		IF DataFromPackML THEN
//			product					:= LREAL_TO_INT(_PackTags.Command.Parameter[2].Value);
//			PullWheels.Length		:= _PackTags.Command.Product[product].ProcessVariables[LENGTH].Value;
//			PullWheels.Velocity		:= _PackTags.Command.Product[product].ProcessVariables[PULLWHEELS_VEL].Value;
//			PullWheels.Acceleration := _PackTags.Command.Product[product].ProcessVariables[PULLWHEELS_ACC].Value;
//			Sealer.SealTime			:= _PackTags.Command.Product[product].ProcessVariables[SEALTIME].Value;
//			Sealer.Temp				:= _PackTags.Command.Product[product].ProcessVariables[SEALTEMP].Value;
//			Sealer.OpenPos			:= _PackTags.Command.Product[product].ProcessVariables[OPEN_POS].Value;
//			Sealer.ClosedPos		:= _PackTags.Command.Product[product].ProcessVariables[CLOSED_POS].Value;
//			Sealer.Velocity			:= _PackTags.Command.Product[product].ProcessVariables[SEALER_VEL].Value;
//			Sealer.Acceleration		:= _PackTags.Command.Product[product].ProcessVariables[SEALER_ACC].Value;
//			Unwind.Velocity			:= _PackTags.Command.Product[product].ProcessVariables[UNWIND_VEL].Value;
//			Unwind.Acceleration		:= _PackTags.Command.Product[product].ProcessVariables[UNWIND_ACC].Value;
		END_IF

	E_PMLUnitMode.ePMLUnitMode_Maintenance, E_PMLUnitMode.ePMLUnitMode_Manual:
		;
END_CASE

SUPER^.Resetting();
END_METHOD

METHOD PROTECTED Starting
VAR_INPUT
END_VAR
CASE _CurrentMode OF
	//=================================PRODUCTION MODE==================================
	E_PMLUnitMode.ePMLUnitMode_Production:
		// The seal bar can go to Execute, the others will be run in Mahcine Execute
	//	Sealer.Heat := TRUE;
		StateComplete();

	E_PMLUnitMode.ePMLUnitMode_Maintenance, E_PMLUnitMode.ePMLUnitMode_Manual:
		SUPER^.Starting();
END_CASE
END_METHOD

METHOD PROTECTED SubModuleMonitor : BOOL
VAR
	AlarmResponses : ARRAY[0..4] OF E_AlarmResponse; //Temporary response array	
END_VAR
// Check the sub Modules for Alarm Severity
SUPER^.SubModuleMonitor();

//Check the alarms at the machine level
_CurrentAlarmSeverity := F_GetMaxSeverityRaised(Alarms := MachineSafetyAlarms, CurrentSeverity := _CurrentAlarmSeverity);

//Check the severity of the machine level alarms
IF _CurrentState <> E_PMLState.ePMLState_Aborted AND _CurrentState <> E_PMLState.ePMLState_Aborting AND _CurrentState <> E_PMLState.ePMLState_Clearing AND _CurrentState <> E_PMLState.ePMLState_Stopped AND _CurrentState <> E_PMLState.ePMLState_Stopping THEN
	AlarmResponses := _ParentFaultResponseDefinitions;
	CASE AlarmResponses[CurrentAlarmSeverity] OF
		E_AlarmResponse.Abort_ImmediateError:
			AbortImmediateError(Name, TRUE);

		E_AlarmResponse.Abort_Immediate:
			AbortImmediate();

		E_AlarmResponse.Stop_Immediate:
			StopImmediate();

		E_AlarmResponse.Stop_Controlled:
			StopControlled();

		E_AlarmResponse.Hold_Immediate:
			HoldImmediate();

		E_AlarmResponse.Suspend_Immediate:
			SuspendImmediate();

		E_AlarmResponse.Suspend_Controlled:
			SuspendControlled();

		E_AlarmResponse.NoResponse:
			;
	END_CASE
ELSIF _CurrentState = E_PMLState.ePMLState_Stopped OR _CurrentState = E_PMLState.ePMLState_Stopping THEN
	AlarmResponses := _ParentFaultResponseDefinitions;
	CASE AlarmResponses[CurrentAlarmSeverity] OF
		E_AlarmResponse.Abort_ImmediateError:
			AbortImmediateError(Name, TRUE);

		E_AlarmResponse.Abort_Immediate:
			AbortImmediate();

		E_AlarmResponse.NoResponse:
			;
	END_CASE
END_IF
END_METHOD

METHOD PROTECTED Suspended
VAR_INPUT
END_VAR
//IF THIS^.Sealer.sealbar.InTempRange THEN
	ChangeState(E_PMLCommand.ePMLCommand_Unsuspend);
//END_IF
END_METHOD

METHOD PROTECTED Suspending
VAR_INPUT
END_VAR
CASE _CurrentMode OF
	//=================================PRODUCTION MODE==================================
	E_PMLUnitMode.ePMLUnitMode_Production:
	//	IF (Sealer.CurrentState = E_PMLState.ePMLState_Complete OR Sealer.CurrentState = E_PMLState.ePMLState_Idle) AND (PullWheels.CurrentState = E_PMLState.ePMLState_Complete OR PullWheels.CurrentState = E_PMLState.ePMLState_Idle) THEN
			StateComplete();
	//	END_IF

	E_PMLUnitMode.ePMLUnitMode_Maintenance, E_PMLUnitMode.ePMLUnitMode_Manual:
		SUPER^.Suspending();
END_CASE
END_METHOD

METHOD PROTECTED Unholding
VAR_INPUT
END_VAR
CASE _CurrentMode OF
	//=================================PRODUCTION MODE==================================
	E_PMLUnitMode.ePMLUnitMode_Production:
		StateComplete();

	E_PMLUnitMode.ePMLUnitMode_Maintenance, E_PMLUnitMode.ePMLUnitMode_Manual:
		SUPER^.Unholding();
END_CASE
END_METHOD

METHOD PROTECTED Unsuspending
VAR_INPUT
END_VAR
CASE _CurrentMode OF
	//=================================PRODUCTION MODE==================================
	E_PMLUnitMode.ePMLUnitMode_Production:
		StateComplete();

	E_PMLUnitMode.ePMLUnitMode_Maintenance, E_PMLUnitMode.ePMLUnitMode_Manual:
		SUPER^.Unsuspending();
END_CASE
END_METHOD

METHOD UpdateModeTimers
VAR
	currentTime	 : T_DCTIME64;
	timeToUpdate : LREAL;
END_VAR

VAR_INST
	lastTime  : T_DCTIME64 := F_GetActualDcTime64();
	lastState : DINT;
	lastMode  : DINT;
END_VAR
IF _PackTags.Status.StateCurrent <> lastState THEN
	MEMSET(ADR(_PackTags.Admin.StateCurrentTime), 0, SIZEOF(_PackTags.Admin.StateCurrentTime));
	lastState := _PackTags.Status.StateCurrent;
END_IF

IF _PackTags.Status.UnitModeCurrent <> lastMode THEN
	MEMSET(ADR(_PackTags.Admin.ModeCurrentTime), 0, SIZEOF(_PackTags.Admin.ModeCurrentTime));
	lastMode := _PackTags.Status.UnitModeCurrent;
END_IF

currentTime := F_GetActualDcTime64();
IF lastTime <> 0 THEN
	timeToUpdate := ULINT_TO_LREAL(currentTime - lastTime) / 1_000_000_000.0;
END_IF

// only seconds get added to the cumulative timers 
IF timeToUpdate > 1 THEN
	_PackTags.Admin.ModeCummulativeTime[_PackTags.Status.UnitModeCurrent]								  := _PackTags.Admin.ModeCummulativeTime[_PackTags.Status.UnitModeCurrent] + LREAL_TO_DINT(timeToUpdate);
	_PackTags.Admin.ModeCurrentTime[_PackTags.Status.UnitModeCurrent]									  := _PackTags.Admin.ModeCurrentTime[_PackTags.Status.UnitModeCurrent] + LREAL_TO_DINT(timeToUpdate);
	_PackTags.Admin.StateCummulativeTime[_PackTags.Status.UnitModeCurrent, _PackTags.Status.StateCurrent] := _PackTags.Admin.StateCummulativeTime[_PackTags.Status.UnitModeCurrent, _PackTags.Status.StateCurrent] + LREAL_TO_DINT(timeToUpdate);
	_PackTags.Admin.StateCurrentTime[_PackTags.Status.UnitModeCurrent, _PackTags.Status.StateCurrent]	  := _PackTags.Admin.StateCurrentTime[_PackTags.Status.UnitModeCurrent, _PackTags.Status.StateCurrent] + LREAL_TO_DINT(timeToUpdate);
	lastTime																							  := currentTime;
END_IF
END_METHOD

END_FUNCTION_BLOCK

// ---- Machine/FB_Systems.TcPOU
FUNCTION_BLOCK FB_Systems EXTENDS FB_PackML_BaseModule // IMPLEMENTS I_ControlsProductionRate
VAR
	// Sub Modules

	
//	Safety			: FB_Safety_Module			:= (Name := 'Safety', LogStateChanges := TRUE);
	Diagnostics		: FB_Diagnostics_Module		:= (Name := 'Diagnostics', LogStateChanges := TRUE);


	// Components

	//Initial List of Components
	ipComponents_Init : ARRAY[1..Parameters_PackML_Base.MAX_NO_OF_COMPONENTS] OF I_ComponentBase := [];

	//Alarms for this module
	SystemAlarms : ARRAY[1..SYTEM_ALARM_COUNT] OF FB_TcAlarm;

	//Current Recipe Name
	CurrentRecipeName : STRING;

	//Get Data From PackML? Else RecipeManager is running
	DataFromPackML : BOOL := TRUE;

	//Data 
	sealTimeStart : ULINT;
	sealTimeEnd	  : ULINT;
	sealingTime	  : LREAL;
	sealTrig	  : R_TRIG;
	pullTimeStart : ULINT;
	pullTimeEnd	  : ULINT;
	pullingTime	  : LREAL;
	pulltrig	  : R_TRIG;
	partTimeStart : ULINT;
	partTimeEnd	  : ULINT;
	partTime	  : LREAL;
	parts		  : DINT;
	product		  : DINT;

	//Pack Tags for System
	{attribute 'OPC.UA.DA' := '1'}
	_PackTags : ST_PackMLv30Ext; //ST_PackMLv30 is obsolete in Tc3_PackML_V2
END_VAR

VAR CONSTANT
	//PackTag parameter IDs
	LENGTH		   : INT := 1;
	SEALTEMP	   : INT := 2;
	SEALTIME	   : INT := 3;
	PULLWHEELS_VEL : INT := 4;
	PULLWHEELS_ACC : INT := 5;
	SEALER_VEL	   : INT := 6;
	SEALER_ACC	   : INT := 7;
	UNWIND_VEL	   : INT := 8;
	UNWIND_ACC	   : INT := 9;
	OPEN_POS	   : INT := 10;
	CLOSED_POS	   : INT := 11;

	//Alarm count constant
	SYTEM_ALARM_COUNT : INT := 6;
END_VAR

// Simulation variables
VAR
	EstopInput	: BOOL;
	LowAirInput : BOOL;
	ErrorInput	: BOOL;
	WarnInput	: BOOL;
	InfoInput	: BOOL;
END_VAR

//This needs to go straight to run mode I did this on the turbine modules
//Stuff for this module
//Maintenance monitoring.
//System communication - Azure - API
//							MQTT
//System times

METHOD PROTECTED Completing
VAR_INPUT
END_VAR
CASE _CurrentMode OF
	//=================================PRODUCTION MODE==================================
	E_PMLUnitMode.ePMLUnitMode_Production:
		StateComplete();

	E_PMLUnitMode.ePMLUnitMode_Maintenance, E_PMLUnitMode.ePMLUnitMode_Manual:
		SUPER^.Completing();
END_CASE
END_METHOD

METHOD PROTECTED CreateEvents
VAR_INPUT
END_VAR
// Add your event creation here
F_CreateAllEventsInClass(Alarms		:= SystemAlarms,
						 ClassSize	:= SIZEOF(TC_Events.VFFSDemo),
						 pInitEvent := ADR(TC_EVENTS.VFFSDemo.InitReferenceEvent),
						 Prefix		:= Name);

// Super call to base
SUPER^.CreateEvents();
END_METHOD

METHOD CyclicLogic
VAR_INPUT
END_VAR
IF NOT _InitComplete THEN
	_InitComplete := Initialize();
	RETURN;
END_IF

SUPER^.CyclicLogic();

// Fill in the PackTags for the machine output
_PackTags.Status.StateCurrent	 := _CurrentState;
_PackTags.Status.UnitModeCurrent := _CurrentMode;
UpdateModeTimers();

//This is just to simulate some IO for alarms
//CyclicLogic_Simulation();
END_METHOD

METHOD CyclicLogic_Simulation
VAR_INPUT
END_VAR

VAR_INST
END_VAR
(*	
This is just for testing. Real hardware can be setup in other places
Here the alarms will raise and clear on its own if the input changes	
*)
IF EstopInput AND NOT MachineAlarms[E_VFFSDemo.EmergencyStop].bRaised THEN
	RaiseAlarm2Args(MachineAlarms[E_VFFSDemo.EmergencyStop], '', '');
ELSIF NOT EstopInput AND MachineAlarms[E_VFFSDemo.EmergencyStop].bRaised THEN
	MachineAlarms[E_VFFSDemo.EmergencyStop].Clear(0, 0);
END_IF

IF LowAirInput AND NOT MachineAlarms[E_VFFSDemo.LowAir].bRaised THEN
	RaiseAlarm2Args(MachineAlarms[E_VFFSDemo.LowAir], '', '');
ELSIF NOT LowAirInput AND MachineAlarms[E_VFFSDemo.LowAir].bRaised THEN
	MachineAlarms[E_VFFSDemo.LowAir].Clear(0, 0);
END_IF

//Generic Alarms for Testing
IF ErrorInput AND NOT MachineAlarms[E_VFFSDemo.AlarmMessage].bRaised THEN
	RaiseAlarm2Args(MachineAlarms[E_VFFSDemo.AlarmMessage], '', '');
ELSIF NOT ErrorInput AND MachineAlarms[E_VFFSDemo.AlarmMessage].bRaised THEN
	MachineAlarms[E_VFFSDemo.AlarmMessage].Clear(0, 0);
END_IF

IF WarnInput AND NOT MachineAlarms[E_VFFSDemo.WarnMessage].bRaised THEN
	RaiseAlarm2Args(MachineAlarms[E_VFFSDemo.WarnMessage], '', '');
ELSIF NOT WarnInput AND MachineAlarms[E_VFFSDemo.WarnMessage].bRaised THEN
	MachineAlarms[E_VFFSDemo.WarnMessage].Clear(0, 0);
END_IF

IF InfoInput AND NOT MachineAlarms[E_VFFSDemo.InfoMessage].bRaised THEN
	RaiseAlarm2Args(MachineAlarms[E_VFFSDemo.InfoMessage], '', '');
ELSIF NOT InfoInput AND MachineAlarms[E_VFFSDemo.InfoMessage].bRaised THEN
	MachineAlarms[E_VFFSDemo.InfoMessage].Clear(0, 0);
END_IF
END_METHOD

METHOD PROTECTED FINAL Execute
VAR_INPUT
END_VAR
CASE _CurrentMode OF
	//=================================PRODUCTION MODE==================================
	E_PMLUnitMode.ePMLUnitMode_Production:
		(* Run the sequence to make products 
		 Unwind Runs Slowly 
		 Pull Wheels Run 
		 Jaws Seal, and Repeat until production reached*)
		sealTrig(CLK := SequenceState = 10);
		IF sealTrig.Q THEN
			partTimeStart := F_GetActualDcTime64();
			sealTimeStart := partTimeStart;
		END_IF

		pulltrig(CLK := SequenceState = 20);
		IF pulltrig.Q THEN
			pullTimeStart := F_GetActualDcTime64();
		END_IF

//		IF THIS^.Sealer.sealbar.InTempRange THEN
//			CASE SequenceState OF
//				0: //Started
//					Unwind.ChangeState(E_PMLCommand.ePMLCommand_Start);
//					IF Unwind.CurrentState = E_PMLState.ePMLState_Execute THEN
//						SequenceState := SequenceState + 10;
//					END_IF

//				10: // SEAL First
//					Sealer.ChangeState(E_PMLCommand.ePMLCommand_Start);
//					IF Sealer.CurrentState = E_PMLState.ePMLState_Complete THEN
//						Sealer.ChangeState(E_PMLCommand.ePMLCommand_Reset);
//						SequenceState := SequenceState + 10;
//						SealTimeEnd	  := F_GetActualDcTime64();
//						sealingTime	  := ULINT_TO_LREAL(sealtimeEnd - sealTimeStart) * 1E-9;
//					END_IF

//				20: // Run Pullwheels
//					PullWheels.ChangeState(E_PMLCommand.ePMLCommand_Start);
//					IF PullWheels.CurrentState = E_PMLState.ePMLState_Complete THEN
//						partTimeEnd	  := F_GetActualDcTime64();
//						parts		  := parts + 1;
//						SequenceState := 10;
//						PullWheels.ChangeState(E_PMLCommand.ePMLCommand_Reset);
//						pullTimeEnd := F_GetActualDcTime64();
//						pullingTime := ULINT_TO_LREAL(pullTimeEnd - pullTimeStart) * 1E-9;
//					END_IF
//			END_CASE
//		ELSE
//			ChangeState(E_PMLCommand.ePMLCommand_Suspend);
//		END_IF

	//=================================MAINTENANCE MODE==================================	
	E_PMLUnitMode.ePMLUnitMode_Maintenance:
		;

	//=================================MANUAL MODE==================================
	E_PMLUnitMode.ePMLUnitMode_Manual:
		;
END_CASE
END_METHOD

METHOD PROTECTED Held
VAR_INPUT
END_VAR
END_METHOD

METHOD PROTECTED HMIPermissions
VAR_INPUT
END_VAR
//General Mode Based Monitoring and handling of HMI control
CASE _CurrentMode OF
	E_PMLUnitMode.ePMLUnitMode_Production:
		CASE _CurrentState OF
			E_PMLState.ePMLState_Stopped:
				AllowHMIControl(ThisModuleOnly := TRUE); //Allow control for recovery
			E_PMLState.ePMLState_Idle:
				//BlockHMIControl();
				AllowHMIControl(ThisModuleOnly := TRUE); //Allow control for recovery
			E_PMLState.ePMLState_Suspended:
				BlockHMIControl();

			E_PMLState.ePMLState_Execute:
				BlockHMIControl();

			E_PMLState.ePMLState_Aborted:
				AllowHMIControl(ThisModuleOnly := TRUE); //Allow control for recovery
			E_PMLState.ePMLState_Held:
				AllowHMIControl(ThisModuleOnly := TRUE); //Allow control for recovery
			E_PMLState.ePMLState_Complete:
				BlockHMIControl();
		END_CASE

	//AllowHMIControl(ThisModuleOnly := FALSE);
	E_PMLUnitMode.ePMLUnitMode_Manual:
		AllowHMIControl(ThisModuleOnly := FALSE);

	E_PMLUnitMode.ePMLUnitMode_Maintenance:
		AllowHMIControl(ThisModuleOnly := FALSE);
END_CASE
END_METHOD

METHOD PROTECTED HoldImmediate
VAR_INPUT
END_VAR
ChangeState(E_PMLCommand.ePMLCommand_Hold);
END_METHOD

METHOD PROTECTED Holding
VAR_INPUT
END_VAR
CASE _CurrentMode OF
	//=================================PRODUCTION MODE==================================
	E_PMLUnitMode.ePMLUnitMode_Production:
	//	IF (Sealer.CurrentState = E_PMLState.ePMLState_Complete OR Sealer.CurrentState = E_PMLState.ePMLState_Idle) AND (PullWheels.CurrentState = E_PMLState.ePMLState_Complete OR PullWheels.CurrentState = E_PMLState.ePMLState_Idle) THEN
			StateComplete();
	//	END_IF

	E_PMLUnitMode.ePMLUnitMode_Maintenance, E_PMLUnitMode.ePMLUnitMode_Manual:
		SUPER^.Holding();
END_CASE
END_METHOD

METHOD PROTECTED Initialize : BOOL
VAR
	i : UDINT; //Generic iteration value
END_VAR
Initialize := FALSE;
CASE DescendantSequenceState OF
	0:
//		RegisterSubmodule(PullWheels);
//		RegisterSubmodule(Sealer);
//		RegisterSubmodule(Unwind);
		
//		RegisterSubmodule(Safety);
		RegisterSubmodule(Diagnostics);
//		RegisterSubmodule(Closer_Gluer);
//		RegisterSubmodule(Labeler);
//		RegisterSubmodule(Diverter);
//		RegisterSubmodule(Outfeed);
		
		_LogModeChanges			:= FALSE;
		_LogStateChanges		:= FALSE;
		DescendantSequenceState := DescendantSequenceState + 10;

	10:
		//Setup Custom modes here

		(*CustomModes(eMode                          :=,
                    sName                          :=,
                    bDisableClearing               :=,
                    bDisableStarting               :=,
                    bDisableSuspended              :=,
                    bDisableStopping               :=,
                    bDisableAborting               :=,
                    bDisableHolding                :=,
                    bDisableHeld                   :=,
                    bDisableUnholding              :=,
                    bDisableSuspending             :=,
                    bDisableUnsuspending           :=,
                    bDisableResetting              :=,
                    bDisableIdle                   :=,
                    bDisableCompleting             :=,
                    bDisableComplete               :=,
                    bEnableUnitModeChangeStopped   :=,
                    bEnableUnitModeChangeIdle      :=,
                    bEnableUnitModeChangeSuspended :=,
                    bEnableUnitModeChangeExecute   :=,
                    bEnableUnitModeChangeAborted   :=,
                    bEnableUnitModeChangeHeld      :=,
                    bEnableUnitModeChangeComplete  :=,
                    bError                         =>,
                    nErrorId                       =>);*)
		DescendantSequenceState := DescendantSequenceState + 10;

	20:
		//Copy Mode names
		FOR i := 1 TO 3 DO
			ModeNames[i] := F_UnitModeToString(UDINT_TO_DINT(i));
		END_FOR

		DescendantSequenceState := DescendantSequenceState + 10;

	30:
		// Initialize Recipes 
		Initialize_Recipes();
		DescendantSequenceState := DescendantSequenceState + 10;

	40:
		//Call the Super
		IF SUPER^.Initialize() THEN
			DescendantSequenceState := DescendantSequenceState + 10;
		END_IF

	50:
		Initialize := TRUE;
END_CASE
END_METHOD

METHOD Initialize_Recipes
VAR_INPUT
END_VAR
// configuration of parameters Max Speed
_packTags.Command.Parameter[1].ID	 := 1;
_packTags.Command.Parameter[1].Name	 := 'Max Speed';
_packTags.Command.Parameter[1].Unit	 := '/min';
_packTags.Command.Parameter[1].Value := 180;
_packTags.Command.Parameter[2].ID	 := 2;
_packTags.Command.Parameter[2].Name	 := 'Product to Run';
_packTags.Command.Parameter[2].Unit	 := '';
_packTags.Command.Parameter[2].Value := 1;

// Recipe Product 1
_PackTags.Command.Product[1].ProductID								:= 100;
_PackTags.Command.Product[1].Ingredients[1].IngredientID			:= 1;
_PackTags.Command.Product[1].Ingredients[1].Parameter[1].ID			:= _PackTags.Command.Product[1].ProductID * 10 + 1;
_PackTags.Command.Product[1].Ingredients[1].Parameter[1].Name		:= 'Material Type';
_PackTags.Command.Product[1].Ingredients[1].Parameter[1].Unit		:= 'n/a';
_PackTags.Command.Product[1].Ingredients[1].Parameter[1].Value		:= 5;
_PackTags.Command.Product[1].Ingredients[1].Parameter[2].ID			:= _PackTags.Command.Product[1].ProductID * 10 + 2;
_PackTags.Command.Product[1].Ingredients[1].Parameter[2].Name		:= 'Material Thickness';
_PackTags.Command.Product[1].Ingredients[1].Parameter[2].Unit		:= 'um';
_PackTags.Command.Product[1].Ingredients[1].Parameter[2].Value		:= 240;
_PackTags.Command.Product[1].ProcessVariables[LENGTH].ID			:= _PackTags.Command.Product[1].ProductID * 20 + 1;
_PackTags.Command.Product[1].ProcessVariables[LENGTH].Name			:= 'Length';
_PackTags.Command.Product[1].ProcessVariables[LENGTH].Unit			:= 'mm';
_PackTags.Command.Product[1].ProcessVariables[LENGTH].Value			:= 100;
_PackTags.Command.Product[1].ProcessVariables[SEALTEMP].ID			:= _PackTags.Command.Product[1].ProductID * 20 + 2;
_PackTags.Command.Product[1].ProcessVariables[SEALTEMP].Name		:= 'Sealing Temp';
_PackTags.Command.Product[1].ProcessVariables[SEALTEMP].Unit		:= 'C';
_PackTags.Command.Product[1].ProcessVariables[SEALTEMP].Value		:= 100;
_PackTags.Command.Product[1].ProcessVariables[SEALTIME].ID			:= _PackTags.Command.Product[1].ProductID * 20 + 3;
_PackTags.Command.Product[1].ProcessVariables[SEALTIME].Name		:= 'Sealing Time';
_PackTags.Command.Product[1].ProcessVariables[SEALTIME].Unit		:= 'ms';
_PackTags.Command.Product[1].ProcessVariables[SEALTIME].Value		:= 50;
_PackTags.Command.Product[1].ProcessVariables[PULLWHEELS_VEL].ID	:= _PackTags.Command.Product[1].ProductID * 20 + 4;
_PackTags.Command.Product[1].ProcessVariables[PULLWHEELS_VEL].Name	:= 'Pull Wheels Vel';
_PackTags.Command.Product[1].ProcessVariables[PULLWHEELS_VEL].Unit	:= 'mm/s';
_PackTags.Command.Product[1].ProcessVariables[PULLWHEELS_VEL].Value := 100;
_PackTags.Command.Product[1].ProcessVariables[PULLWHEELS_ACC].ID	:= _PackTags.Command.Product[1].ProductID * 20 + 5;
_PackTags.Command.Product[1].ProcessVariables[PULLWHEELS_ACC].Name	:= 'Pull Wheels Acc';
_PackTags.Command.Product[1].ProcessVariables[PULLWHEELS_ACC].Unit	:= 'mm/s2';
_PackTags.Command.Product[1].ProcessVariables[PULLWHEELS_ACC].Value := 1000;
_PackTags.Command.Product[1].ProcessVariables[OPEN_POS].ID			:= _PackTags.Command.Product[1].ProductID * 20 + 6;
_PackTags.Command.Product[1].ProcessVariables[OPEN_POS].Name		:= 'Sealer Open Position';
_PackTags.Command.Product[1].ProcessVariables[OPEN_POS].Unit		:= 'mm';
_PackTags.Command.Product[1].ProcessVariables[OPEN_POS].Value		:= 105;
_PackTags.Command.Product[1].ProcessVariables[CLOSED_POS].ID		:= _PackTags.Command.Product[1].ProductID * 20 + 7;
_PackTags.Command.Product[1].ProcessVariables[CLOSED_POS].Name		:= 'Sealer Closed Position';
_PackTags.Command.Product[1].ProcessVariables[CLOSED_POS].Unit		:= 'mm';
_PackTags.Command.Product[1].ProcessVariables[CLOSED_POS].Value		:= 250;
_PackTags.Command.Product[1].ProcessVariables[SEALER_VEL].ID		:= _PackTags.Command.Product[1].ProductID * 20 + 8;
_PackTags.Command.Product[1].ProcessVariables[SEALER_VEL].Name		:= 'Sealer Vel';
_PackTags.Command.Product[1].ProcessVariables[SEALER_VEL].Unit		:= 'mm/s';
_PackTags.Command.Product[1].ProcessVariables[SEALER_VEL].Value		:= 100;
_PackTags.Command.Product[1].ProcessVariables[SEALER_ACC].ID		:= _PackTags.Command.Product[1].ProductID * 20 + 9;
_PackTags.Command.Product[1].ProcessVariables[SEALER_ACC].Name		:= 'Sealer Acc';
_PackTags.Command.Product[1].ProcessVariables[SEALER_ACC].Unit		:= 'mm/s2';
_PackTags.Command.Product[1].ProcessVariables[SEALER_ACC].Value		:= 1000;
_PackTags.Command.Product[1].ProcessVariables[UNWIND_VEL].ID		:= _PackTags.Command.Product[1].ProductID * 20 + 10;
_PackTags.Command.Product[1].ProcessVariables[UNWIND_VEL].Name		:= 'Unwind Vel';
_PackTags.Command.Product[1].ProcessVariables[UNWIND_VEL].Unit		:= 'mm/s';
_PackTags.Command.Product[1].ProcessVariables[UNWIND_VEL].Value		:= 100;
_PackTags.Command.Product[1].ProcessVariables[UNWIND_ACC].ID		:= _PackTags.Command.Product[1].ProductID * 20 + 11;
_PackTags.Command.Product[1].ProcessVariables[UNWIND_ACC].Name		:= 'Unwind Acc';
_PackTags.Command.Product[1].ProcessVariables[UNWIND_ACC].Unit		:= 'mm/s2';
_PackTags.Command.Product[1].ProcessVariables[UNWIND_ACC].Value		:= 1000;

// Product 2
_PackTags.Command.Product[2].ProductID								:= 100;
_PackTags.Command.Product[2].Ingredients[1].IngredientID			:= 1;
_PackTags.Command.Product[2].Ingredients[1].Parameter[1].ID			:= _PackTags.Command.Product[1].ProductID * 10 + 1;
_PackTags.Command.Product[2].Ingredients[1].Parameter[1].Name		:= 'Material Type';
_PackTags.Command.Product[2].Ingredients[1].Parameter[1].Unit		:= 'n/a';
_PackTags.Command.Product[2].Ingredients[1].Parameter[1].Value		:= 2;
_PackTags.Command.Product[2].Ingredients[1].Parameter[2].ID			:= _PackTags.Command.Product[1].ProductID * 10 + 2;
_PackTags.Command.Product[2].Ingredients[1].Parameter[2].Name		:= 'Material Thickness';
_PackTags.Command.Product[2].Ingredients[1].Parameter[2].Unit		:= 'um';
_PackTags.Command.Product[2].Ingredients[1].Parameter[2].Value		:= 220;
_PackTags.Command.Product[2].ProcessVariables[LENGTH].ID			:= _PackTags.Command.Product[1].ProductID * 20 + 1;
_PackTags.Command.Product[2].ProcessVariables[LENGTH].Name			:= 'Length';
_PackTags.Command.Product[2].ProcessVariables[LENGTH].Unit			:= 'mm';
_PackTags.Command.Product[2].ProcessVariables[LENGTH].Value			:= 55;
_PackTags.Command.Product[2].ProcessVariables[SEALTEMP].ID			:= _PackTags.Command.Product[1].ProductID * 20 + 2;
_PackTags.Command.Product[2].ProcessVariables[SEALTEMP].Name		:= 'Sealing Temp';
_PackTags.Command.Product[2].ProcessVariables[SEALTEMP].Unit		:= 'C';
_PackTags.Command.Product[2].ProcessVariables[SEALTEMP].Value		:= 110;
_PackTags.Command.Product[2].ProcessVariables[SEALTIME].ID			:= _PackTags.Command.Product[1].ProductID * 20 + 3;
_PackTags.Command.Product[2].ProcessVariables[SEALTIME].Name		:= 'Sealing Time';
_PackTags.Command.Product[2].ProcessVariables[SEALTIME].Unit		:= 'ms';
_PackTags.Command.Product[2].ProcessVariables[SEALTIME].Value		:= 100;
_PackTags.Command.Product[2].ProcessVariables[PULLWHEELS_VEL].ID	:= _PackTags.Command.Product[1].ProductID * 20 + 4;
_PackTags.Command.Product[2].ProcessVariables[PULLWHEELS_VEL].Name	:= 'Pull Wheels Vel';
_PackTags.Command.Product[2].ProcessVariables[PULLWHEELS_VEL].Unit	:= 'mm/s';
_PackTags.Command.Product[2].ProcessVariables[PULLWHEELS_VEL].Value := 200;
_PackTags.Command.Product[2].ProcessVariables[PULLWHEELS_ACC].ID	:= _PackTags.Command.Product[1].ProductID * 20 + 5;
_PackTags.Command.Product[2].ProcessVariables[PULLWHEELS_ACC].Name	:= 'Pull Wheels Acc';
_PackTags.Command.Product[2].ProcessVariables[PULLWHEELS_ACC].Unit	:= 'mm/s2';
_PackTags.Command.Product[2].ProcessVariables[PULLWHEELS_ACC].Value := 2000;
_PackTags.Command.Product[2].ProcessVariables[OPEN_POS].ID			:= _PackTags.Command.Product[1].ProductID * 20 + 6;
_PackTags.Command.Product[2].ProcessVariables[OPEN_POS].Name		:= 'Sealer Open Position';
_PackTags.Command.Product[2].ProcessVariables[OPEN_POS].Unit		:= 'mm';
_PackTags.Command.Product[2].ProcessVariables[OPEN_POS].Value		:= 60;
_PackTags.Command.Product[2].ProcessVariables[CLOSED_POS].ID		:= _PackTags.Command.Product[1].ProductID * 20 + 7;
_PackTags.Command.Product[2].ProcessVariables[CLOSED_POS].Name		:= 'Sealer Closed Position';
_PackTags.Command.Product[2].ProcessVariables[CLOSED_POS].Unit		:= 'mm';
_PackTags.Command.Product[2].ProcessVariables[CLOSED_POS].Value		:= 253;
_PackTags.Command.Product[2].ProcessVariables[SEALER_VEL].ID		:= _PackTags.Command.Product[1].ProductID * 20 + 8;
_PackTags.Command.Product[2].ProcessVariables[SEALER_VEL].Name		:= 'Sealer Vel';
_PackTags.Command.Product[2].ProcessVariables[SEALER_VEL].Unit		:= 'mm/s';
_PackTags.Command.Product[2].ProcessVariables[SEALER_VEL].Value		:= 200;
_PackTags.Command.Product[2].ProcessVariables[SEALER_ACC].ID		:= _PackTags.Command.Product[1].ProductID * 20 + 9;
_PackTags.Command.Product[2].ProcessVariables[SEALER_ACC].Name		:= 'Sealer Acc';
_PackTags.Command.Product[2].ProcessVariables[SEALER_ACC].Unit		:= 'mm/s2';
_PackTags.Command.Product[2].ProcessVariables[SEALER_ACC].Value		:= 2000;
_PackTags.Command.Product[2].ProcessVariables[UNWIND_VEL].ID		:= _PackTags.Command.Product[1].ProductID * 20 + 10;
_PackTags.Command.Product[2].ProcessVariables[UNWIND_VEL].Name		:= 'Unwind Vel';
_PackTags.Command.Product[2].ProcessVariables[UNWIND_VEL].Unit		:= 'mm/s';
_PackTags.Command.Product[2].ProcessVariables[UNWIND_VEL].Value		:= 200;
_PackTags.Command.Product[2].ProcessVariables[UNWIND_ACC].ID		:= _PackTags.Command.Product[1].ProductID * 20 + 11;
_PackTags.Command.Product[2].ProcessVariables[UNWIND_ACC].Name		:= 'Unwind Acc';
_PackTags.Command.Product[2].ProcessVariables[UNWIND_ACC].Unit		:= 'mm/s2';
_PackTags.Command.Product[2].ProcessVariables[UNWIND_ACC].Value		:= 2000;

//Product 3
_PackTags.Command.Product[3].ProductID								:= 307;
_PackTags.Command.Product[3].Ingredients[1].IngredientID			:= 1;
_PackTags.Command.Product[3].Ingredients[1].Parameter[1].ID			:= _PackTags.Command.Product[1].ProductID * 10 + 1;
_PackTags.Command.Product[3].Ingredients[1].Parameter[1].Name		:= 'Material Type';
_PackTags.Command.Product[3].Ingredients[1].Parameter[1].Unit		:= 'n/a';
_PackTags.Command.Product[3].Ingredients[1].Parameter[1].Value		:= 2;
_PackTags.Command.Product[3].Ingredients[1].Parameter[2].ID			:= _PackTags.Command.Product[1].ProductID * 10 + 2;
_PackTags.Command.Product[3].Ingredients[1].Parameter[2].Name		:= 'Material Thickness';
_PackTags.Command.Product[3].Ingredients[1].Parameter[2].Unit		:= 'um';
_PackTags.Command.Product[3].Ingredients[1].Parameter[2].Value		:= 220;
_PackTags.Command.Product[3].ProcessVariables[LENGTH].ID			:= _PackTags.Command.Product[1].ProductID * 20 + 1;
_PackTags.Command.Product[3].ProcessVariables[LENGTH].Name			:= 'Length';
_PackTags.Command.Product[3].ProcessVariables[LENGTH].Unit			:= 'mm';
_PackTags.Command.Product[3].ProcessVariables[LENGTH].Value			:= 85;
_PackTags.Command.Product[3].ProcessVariables[SEALTEMP].ID			:= _PackTags.Command.Product[1].ProductID * 20 + 2;
_PackTags.Command.Product[3].ProcessVariables[SEALTEMP].Name		:= 'Sealing Temp';
_PackTags.Command.Product[3].ProcessVariables[SEALTEMP].Unit		:= 'C';
_PackTags.Command.Product[3].ProcessVariables[SEALTEMP].Value		:= 95;
_PackTags.Command.Product[3].ProcessVariables[SEALTIME].ID			:= _PackTags.Command.Product[1].ProductID * 20 + 3;
_PackTags.Command.Product[3].ProcessVariables[SEALTIME].Name		:= 'Sealing Time';
_PackTags.Command.Product[3].ProcessVariables[SEALTIME].Unit		:= 'ms';
_PackTags.Command.Product[3].ProcessVariables[SEALTIME].Value		:= 20;
_PackTags.Command.Product[3].ProcessVariables[PULLWHEELS_VEL].ID	:= _PackTags.Command.Product[1].ProductID * 20 + 4;
_PackTags.Command.Product[3].ProcessVariables[PULLWHEELS_VEL].Name	:= 'Pull Wheels Vel';
_PackTags.Command.Product[3].ProcessVariables[PULLWHEELS_VEL].Unit	:= 'mm/s';
_PackTags.Command.Product[3].ProcessVariables[PULLWHEELS_VEL].Value := 300;
_PackTags.Command.Product[3].ProcessVariables[PULLWHEELS_ACC].ID	:= _PackTags.Command.Product[1].ProductID * 20 + 5;
_PackTags.Command.Product[3].ProcessVariables[PULLWHEELS_ACC].Name	:= 'Pull Wheels Acc';
_PackTags.Command.Product[3].ProcessVariables[PULLWHEELS_ACC].Unit	:= 'mm/s2';
_PackTags.Command.Product[3].ProcessVariables[PULLWHEELS_ACC].Value := 3000;
_PackTags.Command.Product[3].ProcessVariables[OPEN_POS].ID			:= _PackTags.Command.Product[1].ProductID * 20 + 6;
_PackTags.Command.Product[3].ProcessVariables[OPEN_POS].Name		:= 'Sealer Open Position';
_PackTags.Command.Product[3].ProcessVariables[OPEN_POS].Unit		:= 'mm';
_PackTags.Command.Product[3].ProcessVariables[OPEN_POS].Value		:= 56;
_PackTags.Command.Product[3].ProcessVariables[CLOSED_POS].ID		:= _PackTags.Command.Product[1].ProductID * 20 + 7;
_PackTags.Command.Product[3].ProcessVariables[CLOSED_POS].Name		:= 'Sealer Closed Position';
_PackTags.Command.Product[3].ProcessVariables[CLOSED_POS].Unit		:= 'mm';
_PackTags.Command.Product[3].ProcessVariables[CLOSED_POS].Value		:= 265;
_PackTags.Command.Product[3].ProcessVariables[SEALER_VEL].ID		:= _PackTags.Command.Product[1].ProductID * 20 + 8;
_PackTags.Command.Product[3].ProcessVariables[SEALER_VEL].Name		:= 'Sealer Vel';
_PackTags.Command.Product[3].ProcessVariables[SEALER_VEL].Unit		:= 'mm/s';
_PackTags.Command.Product[3].ProcessVariables[SEALER_VEL].Value		:= 300;
_PackTags.Command.Product[3].ProcessVariables[SEALER_ACC].ID		:= _PackTags.Command.Product[1].ProductID * 20 + 9;
_PackTags.Command.Product[3].ProcessVariables[SEALER_ACC].Name		:= 'Sealer Acc';
_PackTags.Command.Product[3].ProcessVariables[SEALER_ACC].Unit		:= 'mm/s2';
_PackTags.Command.Product[3].ProcessVariables[SEALER_ACC].Value		:= 3000;
_PackTags.Command.Product[3].ProcessVariables[UNWIND_VEL].ID		:= _PackTags.Command.Product[1].ProductID * 20 + 10;
_PackTags.Command.Product[3].ProcessVariables[UNWIND_VEL].Name		:= 'Unwind Vel';
_PackTags.Command.Product[3].ProcessVariables[UNWIND_VEL].Unit		:= 'mm/s';
_PackTags.Command.Product[3].ProcessVariables[UNWIND_VEL].Value		:= 300;
_PackTags.Command.Product[3].ProcessVariables[UNWIND_ACC].ID		:= _PackTags.Command.Product[1].ProductID * 20 + 11;
_PackTags.Command.Product[3].ProcessVariables[UNWIND_ACC].Name		:= 'Unwind Acc';
_PackTags.Command.Product[3].ProcessVariables[UNWIND_ACC].Unit		:= 'mm/s2';
_PackTags.Command.Product[3].ProcessVariables[UNWIND_ACC].Value		:= 3000;

//Product 4
_PackTags.Command.Product[4].ProductID								:= 401;
_PackTags.Command.Product[4].Ingredients[1].IngredientID			:= 1;
_PackTags.Command.Product[4].Ingredients[1].Parameter[1].ID			:= _PackTags.Command.Product[1].ProductID * 10 + 1;
_PackTags.Command.Product[4].Ingredients[1].Parameter[1].Name		:= 'Material Type';
_PackTags.Command.Product[4].Ingredients[1].Parameter[1].Unit		:= 'n/a';
_PackTags.Command.Product[4].Ingredients[1].Parameter[1].Value		:= 2;
_PackTags.Command.Product[4].Ingredients[1].Parameter[2].ID			:= _PackTags.Command.Product[1].ProductID * 10 + 2;
_PackTags.Command.Product[4].Ingredients[1].Parameter[2].Name		:= 'Material Thickness';
_PackTags.Command.Product[4].Ingredients[1].Parameter[2].Unit		:= 'um';
_PackTags.Command.Product[4].Ingredients[1].Parameter[2].Value		:= 220;
_PackTags.Command.Product[4].ProcessVariables[LENGTH].ID			:= _PackTags.Command.Product[1].ProductID * 20 + 1;
_PackTags.Command.Product[4].ProcessVariables[LENGTH].Name			:= 'Length';
_PackTags.Command.Product[4].ProcessVariables[LENGTH].Unit			:= 'mm';
_PackTags.Command.Product[4].ProcessVariables[LENGTH].Value			:= 85;
_PackTags.Command.Product[4].ProcessVariables[SEALTEMP].ID			:= _PackTags.Command.Product[1].ProductID * 20 + 2;
_PackTags.Command.Product[4].ProcessVariables[SEALTEMP].Name		:= 'Sealing Temp';
_PackTags.Command.Product[4].ProcessVariables[SEALTEMP].Unit		:= 'C';
_PackTags.Command.Product[4].ProcessVariables[SEALTEMP].Value		:= 95;
_PackTags.Command.Product[4].ProcessVariables[SEALTIME].ID			:= _PackTags.Command.Product[1].ProductID * 20 + 3;
_PackTags.Command.Product[4].ProcessVariables[SEALTIME].Name		:= 'Sealing Time';
_PackTags.Command.Product[4].ProcessVariables[SEALTIME].Unit		:= 'ms';
_PackTags.Command.Product[4].ProcessVariables[SEALTIME].Value		:= 80;
_PackTags.Command.Product[4].ProcessVariables[PULLWHEELS_VEL].ID	:= _PackTags.Command.Product[1].ProductID * 20 + 4;
_PackTags.Command.Product[4].ProcessVariables[PULLWHEELS_VEL].Name	:= 'Pull Wheels Vel';
_PackTags.Command.Product[4].ProcessVariables[PULLWHEELS_VEL].Unit	:= 'mm/s';
_PackTags.Command.Product[4].ProcessVariables[PULLWHEELS_VEL].Value := 100;
_PackTags.Command.Product[4].ProcessVariables[PULLWHEELS_ACC].ID	:= _PackTags.Command.Product[1].ProductID * 20 + 5;
_PackTags.Command.Product[4].ProcessVariables[PULLWHEELS_ACC].Name	:= 'Pull Wheels Acc';
_PackTags.Command.Product[4].ProcessVariables[PULLWHEELS_ACC].Unit	:= 'mm/s2';
_PackTags.Command.Product[4].ProcessVariables[PULLWHEELS_ACC].Value := 1000;
_PackTags.Command.Product[4].ProcessVariables[OPEN_POS].ID			:= _PackTags.Command.Product[1].ProductID * 20 + 6;
_PackTags.Command.Product[4].ProcessVariables[OPEN_POS].Name		:= 'Sealer Open Position';
_PackTags.Command.Product[4].ProcessVariables[OPEN_POS].Unit		:= 'mm';
_PackTags.Command.Product[4].ProcessVariables[OPEN_POS].Value		:= 105;
_PackTags.Command.Product[4].ProcessVariables[CLOSED_POS].ID		:= _PackTags.Command.Product[1].ProductID * 20 + 7;
_PackTags.Command.Product[4].ProcessVariables[CLOSED_POS].Name		:= 'Sealer Closed Position';
_PackTags.Command.Product[4].ProcessVariables[CLOSED_POS].Unit		:= 'mm';
_PackTags.Command.Product[4].ProcessVariables[CLOSED_POS].Value		:= 250;
_PackTags.Command.Product[4].ProcessVariables[SEALER_VEL].ID		:= _PackTags.Command.Product[1].ProductID * 20 + 8;
_PackTags.Command.Product[4].ProcessVariables[SEALER_VEL].Name		:= 'Sealer Vel';
_PackTags.Command.Product[4].ProcessVariables[SEALER_VEL].Unit		:= 'mm/s';
_PackTags.Command.Product[4].ProcessVariables[SEALER_VEL].Value		:= 100;
_PackTags.Command.Product[4].ProcessVariables[SEALER_ACC].ID		:= _PackTags.Command.Product[1].ProductID * 20 + 9;
_PackTags.Command.Product[4].ProcessVariables[SEALER_ACC].Name		:= 'Sealer Acc';
_PackTags.Command.Product[4].ProcessVariables[SEALER_ACC].Unit		:= 'mm/s2';
_PackTags.Command.Product[4].ProcessVariables[SEALER_ACC].Value		:= 1000;
_PackTags.Command.Product[4].ProcessVariables[UNWIND_VEL].ID		:= _PackTags.Command.Product[1].ProductID * 20 + 10;
_PackTags.Command.Product[4].ProcessVariables[UNWIND_VEL].Name		:= 'Unwind Vel';
_PackTags.Command.Product[4].ProcessVariables[UNWIND_VEL].Unit		:= 'mm/s';
_PackTags.Command.Product[4].ProcessVariables[UNWIND_VEL].Value		:= 100;
_PackTags.Command.Product[4].ProcessVariables[UNWIND_ACC].ID		:= _PackTags.Command.Product[1].ProductID * 20 + 11;
_PackTags.Command.Product[4].ProcessVariables[UNWIND_ACC].Name		:= 'Unwind Acc';
_PackTags.Command.Product[4].ProcessVariables[UNWIND_ACC].Unit		:= 'mm/s2';
_PackTags.Command.Product[4].ProcessVariables[UNWIND_ACC].Value		:= 1000;

//Product 5
_PackTags.Command.Product[5].ProductID								:= 522;
_PackTags.Command.Product[5].Ingredients[1].IngredientID			:= 1;
_PackTags.Command.Product[5].Ingredients[1].Parameter[1].ID			:= _PackTags.Command.Product[1].ProductID * 10 + 1;
_PackTags.Command.Product[5].Ingredients[1].Parameter[1].Name		:= 'Material Type';
_PackTags.Command.Product[5].Ingredients[1].Parameter[1].Unit		:= 'n/a';
_PackTags.Command.Product[5].Ingredients[1].Parameter[1].Value		:= 2;
_PackTags.Command.Product[5].Ingredients[1].Parameter[2].ID			:= _PackTags.Command.Product[1].ProductID * 10 + 2;
_PackTags.Command.Product[5].Ingredients[1].Parameter[2].Name		:= 'Material Thickness';
_PackTags.Command.Product[5].Ingredients[1].Parameter[2].Unit		:= 'um';
_PackTags.Command.Product[5].Ingredients[1].Parameter[2].Value		:= 520;
_PackTags.Command.Product[5].ProcessVariables[LENGTH].ID			:= _PackTags.Command.Product[1].ProductID * 20 + 1;
_PackTags.Command.Product[5].ProcessVariables[LENGTH].Name			:= 'Length';
_PackTags.Command.Product[5].ProcessVariables[LENGTH].Unit			:= 'mm';
_PackTags.Command.Product[5].ProcessVariables[LENGTH].Value			:= 200;
_PackTags.Command.Product[5].ProcessVariables[SEALTEMP].ID			:= _PackTags.Command.Product[1].ProductID * 20 + 2;
_PackTags.Command.Product[5].ProcessVariables[SEALTEMP].Name		:= 'Sealing Temp';
_PackTags.Command.Product[5].ProcessVariables[SEALTEMP].Unit		:= 'C';
_PackTags.Command.Product[5].ProcessVariables[SEALTEMP].Value		:= 130;
_PackTags.Command.Product[5].ProcessVariables[SEALTIME].ID			:= _PackTags.Command.Product[1].ProductID * 20 + 3;
_PackTags.Command.Product[5].ProcessVariables[SEALTIME].Name		:= 'Sealing Time';
_PackTags.Command.Product[5].ProcessVariables[SEALTIME].Unit		:= 'ms';
_PackTags.Command.Product[5].ProcessVariables[SEALTIME].Value		:= 200;
_PackTags.Command.Product[5].ProcessVariables[PULLWHEELS_VEL].ID	:= _PackTags.Command.Product[1].ProductID * 20 + 4;
_PackTags.Command.Product[5].ProcessVariables[PULLWHEELS_VEL].Name	:= 'Pull Wheels Vel';
_PackTags.Command.Product[5].ProcessVariables[PULLWHEELS_VEL].Unit	:= 'mm/s';
_PackTags.Command.Product[5].ProcessVariables[PULLWHEELS_VEL].Value := 100;
_PackTags.Command.Product[5].ProcessVariables[PULLWHEELS_ACC].ID	:= _PackTags.Command.Product[1].ProductID * 20 + 5;
_PackTags.Command.Product[5].ProcessVariables[PULLWHEELS_ACC].Name	:= 'Pull Wheels Acc';
_PackTags.Command.Product[5].ProcessVariables[PULLWHEELS_ACC].Unit	:= 'mm/s2';
_PackTags.Command.Product[5].ProcessVariables[PULLWHEELS_ACC].Value := 1000;
_PackTags.Command.Product[5].ProcessVariables[OPEN_POS].ID			:= _PackTags.Command.Product[1].ProductID * 20 + 6;
_PackTags.Command.Product[5].ProcessVariables[OPEN_POS].Name		:= 'Sealer Open Position';
_PackTags.Command.Product[5].ProcessVariables[OPEN_POS].Unit		:= 'mm';
_PackTags.Command.Product[5].ProcessVariables[OPEN_POS].Value		:= 105;
_PackTags.Command.Product[5].ProcessVariables[CLOSED_POS].ID		:= _PackTags.Command.Product[1].ProductID * 20 + 7;
_PackTags.Command.Product[5].ProcessVariables[CLOSED_POS].Name		:= 'Sealer Closed Position';
_PackTags.Command.Product[5].ProcessVariables[CLOSED_POS].Unit		:= 'mm';
_PackTags.Command.Product[5].ProcessVariables[CLOSED_POS].Value		:= 250;
_PackTags.Command.Product[5].ProcessVariables[SEALER_VEL].ID		:= _PackTags.Command.Product[1].ProductID * 20 + 8;
_PackTags.Command.Product[5].ProcessVariables[SEALER_VEL].Name		:= 'Sealer Vel';
_PackTags.Command.Product[5].ProcessVariables[SEALER_VEL].Unit		:= 'mm/s';
_PackTags.Command.Product[5].ProcessVariables[SEALER_VEL].Value		:= 100;
_PackTags.Command.Product[5].ProcessVariables[SEALER_ACC].ID		:= _PackTags.Command.Product[1].ProductID * 20 + 9;
_PackTags.Command.Product[5].ProcessVariables[SEALER_ACC].Name		:= 'Sealer Acc';
_PackTags.Command.Product[5].ProcessVariables[SEALER_ACC].Unit		:= 'mm/s2';
_PackTags.Command.Product[5].ProcessVariables[SEALER_ACC].Value		:= 1000;
_PackTags.Command.Product[5].ProcessVariables[UNWIND_VEL].ID		:= _PackTags.Command.Product[1].ProductID * 20 + 10;
_PackTags.Command.Product[5].ProcessVariables[UNWIND_VEL].Name		:= 'Unwind Vel';
_PackTags.Command.Product[5].ProcessVariables[UNWIND_VEL].Unit		:= 'mm/s';
_PackTags.Command.Product[5].ProcessVariables[UNWIND_VEL].Value		:= 100;
_PackTags.Command.Product[5].ProcessVariables[UNWIND_ACC].ID		:= _PackTags.Command.Product[1].ProductID * 20 + 11;
_PackTags.Command.Product[5].ProcessVariables[UNWIND_ACC].Name		:= 'Unwind Acc';
_PackTags.Command.Product[5].ProcessVariables[UNWIND_ACC].Unit		:= 'mm/s2';
_PackTags.Command.Product[5].ProcessVariables[UNWIND_ACC].Value		:= 1000;
CurrentRecipeName													:= 'From PackTags';
END_METHOD

PROPERTY PUBLIC PackTags : ST_PackMLv30Ext
GET
PackTags := _packTags;
END_GET
END_PROPERTY

METHOD RaiseAlarm2Args
VAR_IN_OUT
	Alarm : FB_TcAlarm; //Alarm to be raised
END_VAR

VAR_INPUT
	String_1 : STRING; //First String Parameter (The Name of this component will be applied first automatically)
	String_2 : STRING; //Second String Parameter
END_VAR
F_RaiseAlarmWithStringParameters(Alarm	  := Alarm,
								 String_1 := Name,
								 String_2 := String_1,
								 String_3 := String_2);
END_METHOD

METHOD PROTECTED Resetting
VAR_INPUT
END_VAR
CASE _CurrentMode OF
	//=================================PRODUCTION MODE==================================
	E_PMLUnitMode.ePMLUnitMode_Production:
		IF DataFromPackML THEN
			product					:= LREAL_TO_INT(_PackTags.Command.Parameter[2].Value);
//			PullWheels.Length		:= _PackTags.Command.Product[product].ProcessVariables[LENGTH].Value;
//			PullWheels.Velocity		:= _PackTags.Command.Product[product].ProcessVariables[PULLWHEELS_VEL].Value;
//			PullWheels.Acceleration := _PackTags.Command.Product[product].ProcessVariables[PULLWHEELS_ACC].Value;
//			Sealer.SealTime			:= _PackTags.Command.Product[product].ProcessVariables[SEALTIME].Value;
//			Sealer.Temp				:= _PackTags.Command.Product[product].ProcessVariables[SEALTEMP].Value;
//			Sealer.OpenPos			:= _PackTags.Command.Product[product].ProcessVariables[OPEN_POS].Value;
//			Sealer.ClosedPos		:= _PackTags.Command.Product[product].ProcessVariables[CLOSED_POS].Value;
//			Sealer.Velocity			:= _PackTags.Command.Product[product].ProcessVariables[SEALER_VEL].Value;
//			Sealer.Acceleration		:= _PackTags.Command.Product[product].ProcessVariables[SEALER_ACC].Value;
//			Unwind.Velocity			:= _PackTags.Command.Product[product].ProcessVariables[UNWIND_VEL].Value;
//			Unwind.Acceleration		:= _PackTags.Command.Product[product].ProcessVariables[UNWIND_ACC].Value;
		END_IF

	E_PMLUnitMode.ePMLUnitMode_Maintenance, E_PMLUnitMode.ePMLUnitMode_Manual:
		;
END_CASE

SUPER^.Resetting();
END_METHOD

METHOD PROTECTED Starting
VAR_INPUT
END_VAR
CASE _CurrentMode OF
	//=================================PRODUCTION MODE==================================
	E_PMLUnitMode.ePMLUnitMode_Production:
		// The seal bar can go to Execute, the others will be run in Mahcine Execute
	//	Sealer.Heat := TRUE;
		StateComplete();

	E_PMLUnitMode.ePMLUnitMode_Maintenance, E_PMLUnitMode.ePMLUnitMode_Manual:
		SUPER^.Starting();
END_CASE
END_METHOD

METHOD PROTECTED SubModuleMonitor : BOOL
VAR
	AlarmResponses : ARRAY[0..4] OF E_AlarmResponse; //Temporary response array	
END_VAR
// Check the sub Modules for Alarm Severity
SUPER^.SubModuleMonitor();

//Check the alarms at the machine level
_CurrentAlarmSeverity := F_GetMaxSeverityRaised(Alarms := SystemAlarms, CurrentSeverity := _CurrentAlarmSeverity);

//Check the severity of the machine level alarms
IF _CurrentState <> E_PMLState.ePMLState_Aborted AND _CurrentState <> E_PMLState.ePMLState_Aborting AND _CurrentState <> E_PMLState.ePMLState_Clearing AND _CurrentState <> E_PMLState.ePMLState_Stopped AND _CurrentState <> E_PMLState.ePMLState_Stopping THEN
	AlarmResponses := _ParentFaultResponseDefinitions;
	CASE AlarmResponses[CurrentAlarmSeverity] OF
		E_AlarmResponse.Abort_ImmediateError:
			AbortImmediateError(Name, TRUE);

		E_AlarmResponse.Abort_Immediate:
			AbortImmediate();

		E_AlarmResponse.Stop_Immediate:
			StopImmediate();

		E_AlarmResponse.Stop_Controlled:
			StopControlled();

		E_AlarmResponse.Hold_Immediate:
			HoldImmediate();

		E_AlarmResponse.Suspend_Immediate:
			SuspendImmediate();

		E_AlarmResponse.Suspend_Controlled:
			SuspendControlled();

		E_AlarmResponse.NoResponse:
			;
	END_CASE
ELSIF _CurrentState = E_PMLState.ePMLState_Stopped OR _CurrentState = E_PMLState.ePMLState_Stopping THEN
	AlarmResponses := _ParentFaultResponseDefinitions;
	CASE AlarmResponses[CurrentAlarmSeverity] OF
		E_AlarmResponse.Abort_ImmediateError:
			AbortImmediateError(Name, TRUE);

		E_AlarmResponse.Abort_Immediate:
			AbortImmediate();

		E_AlarmResponse.NoResponse:
			;
	END_CASE
END_IF
END_METHOD

METHOD PROTECTED Suspended
VAR_INPUT
END_VAR
//IF THIS^.Sealer.sealbar.InTempRange THEN
	ChangeState(E_PMLCommand.ePMLCommand_Unsuspend);
//END_IF
END_METHOD

METHOD PROTECTED Suspending
VAR_INPUT
END_VAR
CASE _CurrentMode OF
	//=================================PRODUCTION MODE==================================
	E_PMLUnitMode.ePMLUnitMode_Production:
	//	IF (Sealer.CurrentState = E_PMLState.ePMLState_Complete OR Sealer.CurrentState = E_PMLState.ePMLState_Idle) AND (PullWheels.CurrentState = E_PMLState.ePMLState_Complete OR PullWheels.CurrentState = E_PMLState.ePMLState_Idle) THEN
			StateComplete();
	//	END_IF

	E_PMLUnitMode.ePMLUnitMode_Maintenance, E_PMLUnitMode.ePMLUnitMode_Manual:
		SUPER^.Suspending();
END_CASE
END_METHOD

METHOD PROTECTED Unholding
VAR_INPUT
END_VAR
CASE _CurrentMode OF
	//=================================PRODUCTION MODE==================================
	E_PMLUnitMode.ePMLUnitMode_Production:
		StateComplete();

	E_PMLUnitMode.ePMLUnitMode_Maintenance, E_PMLUnitMode.ePMLUnitMode_Manual:
		SUPER^.Unholding();
END_CASE
END_METHOD

METHOD PROTECTED Unsuspending
VAR_INPUT
END_VAR
CASE _CurrentMode OF
	//=================================PRODUCTION MODE==================================
	E_PMLUnitMode.ePMLUnitMode_Production:
		StateComplete();

	E_PMLUnitMode.ePMLUnitMode_Maintenance, E_PMLUnitMode.ePMLUnitMode_Manual:
		SUPER^.Unsuspending();
END_CASE
END_METHOD

METHOD UpdateModeTimers
VAR
	currentTime	 : T_DCTIME64;
	timeToUpdate : LREAL;
END_VAR

VAR_INST
	lastTime  : T_DCTIME64 := F_GetActualDcTime64();
	lastState : DINT;
	lastMode  : DINT;
END_VAR
IF _PackTags.Status.StateCurrent <> lastState THEN
	MEMSET(ADR(_PackTags.Admin.StateCurrentTime), 0, SIZEOF(_PackTags.Admin.StateCurrentTime));
	lastState := _PackTags.Status.StateCurrent;
END_IF

IF _PackTags.Status.UnitModeCurrent <> lastMode THEN
	MEMSET(ADR(_PackTags.Admin.ModeCurrentTime), 0, SIZEOF(_PackTags.Admin.ModeCurrentTime));
	lastMode := _PackTags.Status.UnitModeCurrent;
END_IF

currentTime := F_GetActualDcTime64();
IF lastTime <> 0 THEN
	timeToUpdate := ULINT_TO_LREAL(currentTime - lastTime) / 1_000_000_000.0;
END_IF

// only seconds get added to the cumulative timers 
IF timeToUpdate > 1 THEN
	_PackTags.Admin.ModeCummulativeTime[_PackTags.Status.UnitModeCurrent]								  := _PackTags.Admin.ModeCummulativeTime[_PackTags.Status.UnitModeCurrent] + LREAL_TO_DINT(timeToUpdate);
	_PackTags.Admin.ModeCurrentTime[_PackTags.Status.UnitModeCurrent]									  := _PackTags.Admin.ModeCurrentTime[_PackTags.Status.UnitModeCurrent] + LREAL_TO_DINT(timeToUpdate);
	_PackTags.Admin.StateCummulativeTime[_PackTags.Status.UnitModeCurrent, _PackTags.Status.StateCurrent] := _PackTags.Admin.StateCummulativeTime[_PackTags.Status.UnitModeCurrent, _PackTags.Status.StateCurrent] + LREAL_TO_DINT(timeToUpdate);
	_PackTags.Admin.StateCurrentTime[_PackTags.Status.UnitModeCurrent, _PackTags.Status.StateCurrent]	  := _PackTags.Admin.StateCurrentTime[_PackTags.Status.UnitModeCurrent, _PackTags.Status.StateCurrent] + LREAL_TO_DINT(timeToUpdate);
	lastTime																							  := currentTime;
END_IF
END_METHOD

END_FUNCTION_BLOCK

// ---- GlobalTextList.TcGTLO
TEXTLIST GlobalTextList
  733 = '%0.1f °'
  282 = '%d'
  685 = '%s'
  680 = 'Abort'
  452 = 'Clear'
  809 = 'Clear Unwind'
  424 = 'EStop'
  408 = 'EtherCat Master'
  744 = 'Hold'
  194 = 'ID:'
  517 = 'Low Air'
  347 = 'MACHINE'
  46 = 'Maintenance'
  904 = 'Manual'
  929 = 'Production'
  181 = 'Reset'
  538 = 'Reset Unwind'
  54 = 'SAFETY'
  206 = 'Simulate \nAll'
  436 = 'Simulate All'
  77 = 'Start'
  804 = 'Start Unwind'
  963 = 'State: %d'
  516 = 'State: %s'
  828 = 'Stop'
  806 = 'Suspend'
  995 = 'Temp Setpoint'
  197 = 'Unhold'
  832 = 'Unsuspend'
END_TEXTLIST

// ---- Machine/VISUs/VisuOjects/V_EtherCatMasterComponent.TcVIS
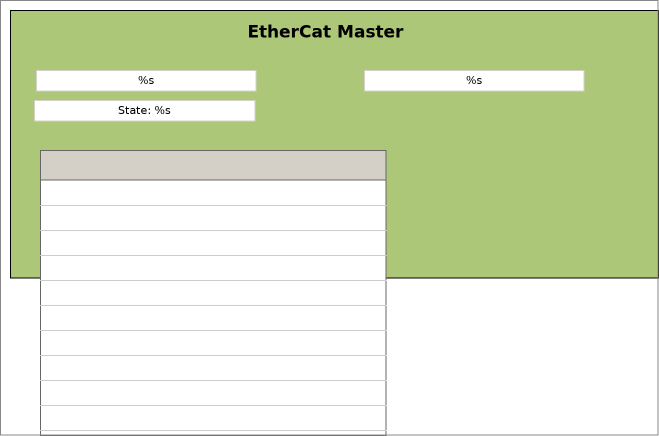
VISUALIZATION V_EtherCatMasterComponent  // 659x436
VAR_IN_OUT
	EtherCatMaster_HMI : ST_EtherCatMaster_HMI;
END_VAR
(*
		AmsNetID			: T_AMSNETID;
		CfgSlaveCount		: UINT;
		EcSlavesState		: ARRAY[0..EC_MAX_SLAVES] OF ST_EcSlaveState;
		ConfiguredSlaveInfo : ARRAY[0..EC_MAX_SLAVES] OF ST_EcSlaveConfigData;
		EcSlaveTopologyInfo : ARRAY[0..EC_MAX_SLAVES] OF ST_TopologyDataEx;
*)
    RoundedRectangle (10,10 649x268)
    Label (41,13 569x37), "EtherCat Master"
    Textfield (34,100 221x21), "State: %s", text variable: HMI.Status.State
    Textfield (36,70 220x21), "%s", text variable: EtherCatMaster_HMI.Status.
    Table (40,150 346x286)
    Textfield (364,70 220x21), "%s", text variable: EtherCatMaster_HMI.Status.ConfiguredSlaveInfo
END_VISUALIZATION

// ---- Machine/VISUs/VisuOjects/V_MachineModule.TcVIS
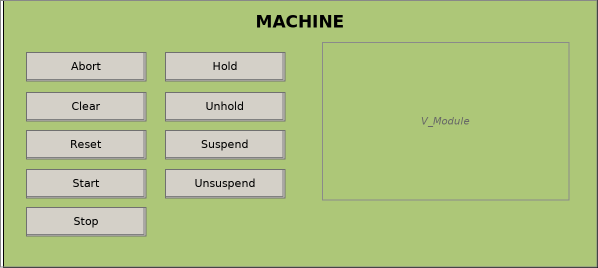
VISUALIZATION V_MachineModule  // 598x268
VAR_IN_OUT
	HMI : ST_PackMLBaseModule_HMI;
END_VAR
    Group (3,0 595x268)
        RoundedRectangle (0,0 595x268)
        Button (23,52 120x29), "Abort"
            OnMouseClick: execute { HMI.Command.State := E_PMLCommand.ePMLCommand_Abort; }
        Button (23,92 120x29), "Clear"
            OnMouseClick: execute { HMI.Command.State := E_PMLCommand.ePMLCommand_Clear; }
        Button (23,130 120x29), "Reset"
            OnMouseClick: execute { HMI.Command.State := E_PMLCommand.ePMLCommand_Reset; }
        Button (23,169 120x29), "Start"
            OnMouseClick: execute { HMI.Command.State := E_PMLCommand.ePMLCommand_Start; }
        Button (23,207 120x29), "Stop"
            OnMouseClick: execute { HMI.Command.State := E_PMLCommand.ePMLCommand_Stop; }
        Button (162,52 120x29), "Hold"
            OnMouseClick: execute { HMI.Command.State := E_PMLCommand.ePMLCommand_Hold; }
        Button (162,92 120x29), "Unhold"
            OnMouseClick: execute { HMI.Command.State := E_PMLCommand.ePMLCommand_Unhold; }
        Button (162,130 120x29), "Suspend"
            OnMouseClick: execute { HMI.Command.State := E_PMLCommand.ePMLCommand_Suspend; }
        Button (162,169 120x29), "Unsuspend"
            OnMouseClick: execute { HMI.Command.State := E_PMLCommand.ePMLCommand_Unsuspend; }
        Frame (319,42 247x158)
            shows V_Module(HMI := HMI)
    Label (15,3 570x37), "MACHINE"
END_VISUALIZATION

// ---- Machine/VISUs/VisuOjects/V_SafetyModule.TcVIS
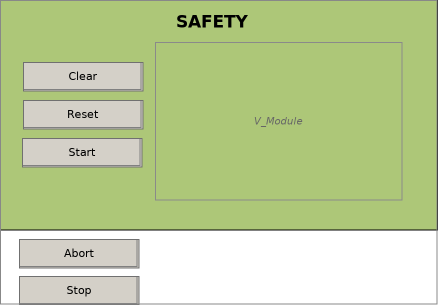
VISUALIZATION V_SafetyModule  // 438x305
VAR_IN_OUT
	HMI : ST_PackMLBaseModule_HMI;
END_VAR
    RoundedRectangle (0,0 438x230)
    Button (19,239 120x29), "Abort"
        OnMouseClick: execute { HMI.Command.State := E_PMLCommand.ePMLCommand_Abort; }
    Button (23,62 120x29), "Clear"
        OnMouseClick: execute { HMI.Command.State := E_PMLCommand.ePMLCommand_Clear; }
    Button (23,100 120x29), "Reset"
        OnMouseClick: execute { HMI.Command.State := E_PMLCommand.ePMLCommand_Reset; }
    Button (22,138 120x29), "Start"
        OnMouseClick: execute { HMI.Command.State := E_PMLCommand.ePMLCommand_Start; }
    Button (19,276 120x29), "Stop"
        OnMouseClick: execute { HMI.Command.State := E_PMLCommand.ePMLCommand_Stop; }
    Frame (155,42 247x158)
        shows V_Module(HMI := HMI)
    Label (31,3 362x37), "SAFETY"
END_VISUALIZATION

// ---- Machine/VISUs/V_Main.TcVIS
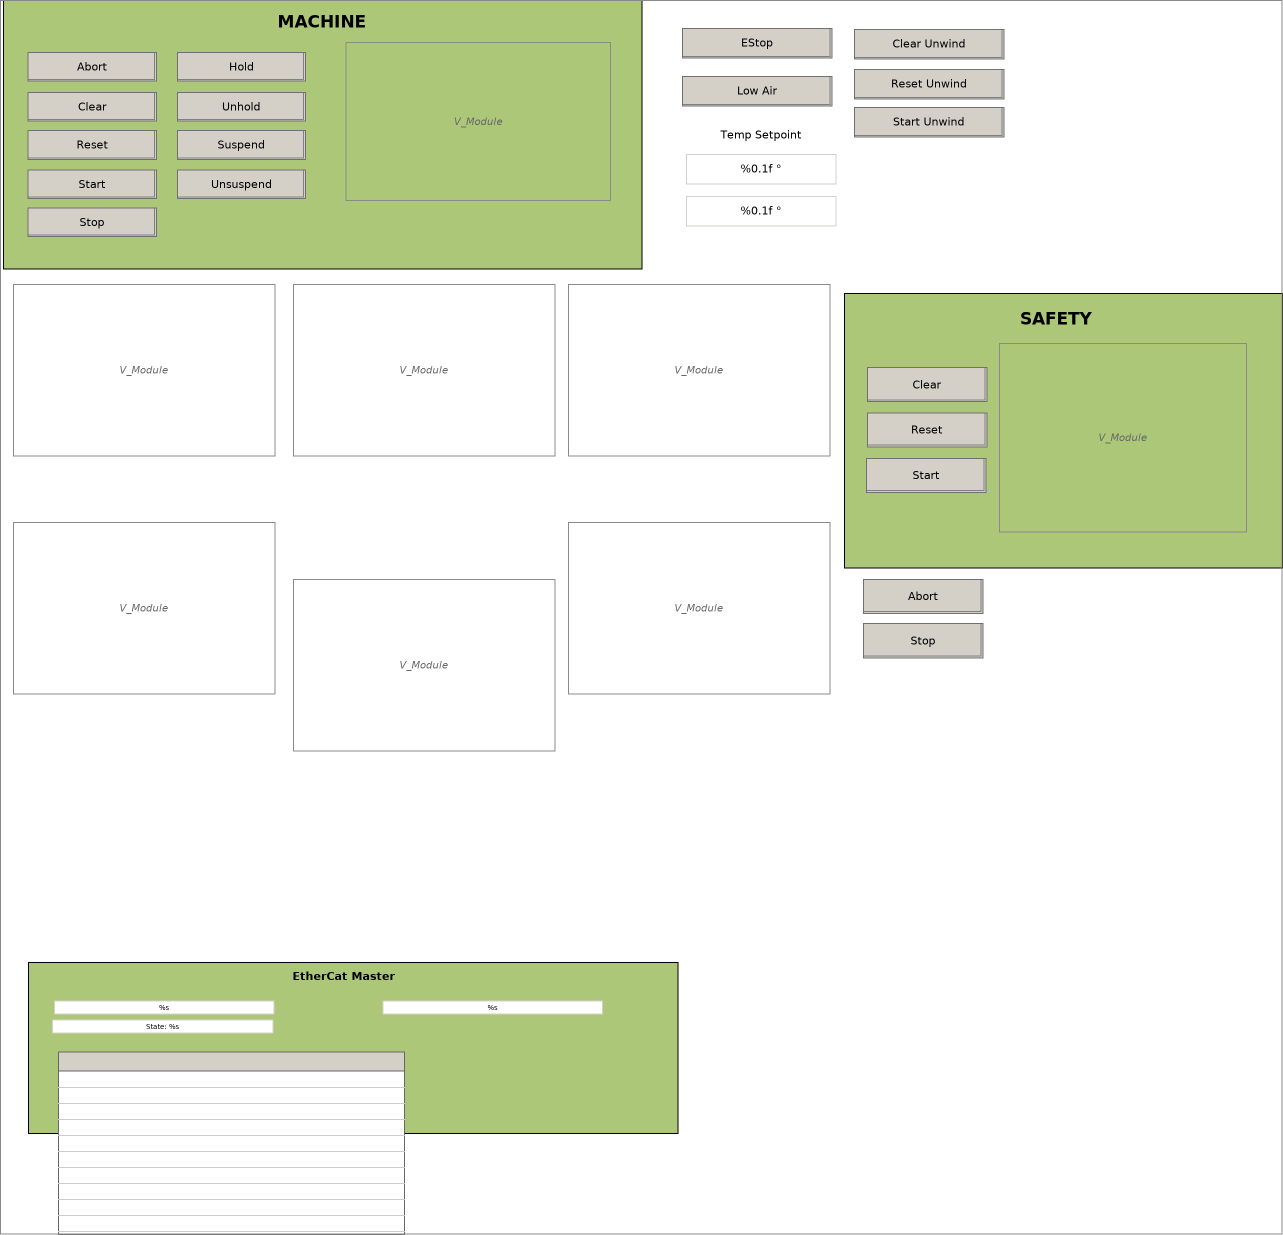
VISUALIZATION V_Main  // 1283x1235
    Frame (0,0 642x269)
        shows V_MachineModule(HMI := MAIN.Machine.PackMLBaseModule_HMI)
    Frame (568,284 262x172)
        shows V_Module(HMI := MAIN.Machine.Station_4.PackMLBaseModule_HMI)
    Frame (568,522 262x172)
        shows V_Module(HMI := MAIN.Machine.Station_5.PackMLBaseModule_HMI)
    Button (682,28 150x30), "EStop"
        toggle MAIN.Machine.EstopInput
    Button (682,76 150x30), "Low Air"
        toggle MAIN.Machine.LowAirInput
    Textfield (686,154 150x30), "%0.1f °", text variable: MAIN.Machine.Sealer.SealBar._SetTemperature
        OnMouseDown: write the text variable via VisuDialogs.Numpad, min 20, max 400, title 'Sealer Bar Temp Setpoint', format %0.1f
    Label (686,120 150x30), "Temp Setpoint"
    Textfield (686,196 150x30), "%0.1f °", text variable: MAIN.Machine.Sealer.SealBar._ActualTemperature
    Button (854,29 150x30), "Clear Unwind"
        OnMouseClick: execute { MAIN.Machine.unwind.PackMLBaseModule_HMI.Command.State := E_PMLCommand.ePMLCommand_Clear; }
    Button (854,69 150x30), "Reset Unwind"
        OnMouseClick: execute { MAIN.Machine.unwind.PackMLBaseModule_HMI.Command.State := E_PMLCommand.ePMLCommand_Reset; }
    Button (854,107 150x30), "Start Unwind"
        OnMouseClick: execute { MAIN.Machine.unwind.PackMLBaseModule_HMI.Command.State := E_PMLCommand.ePMLCommand_Start; }
    Frame (844,293 439x365)
        shows V_SafetyModule(HMI := MAIN.Machine.Safety_SubModule.PackMLBaseModule_HMI)
    Frame (18,956 660x279)
        shows V_EtherCatMasterComponent(EtherCatMaster_HMI := MAIN.Machine.Systems_SubModule.Diagnostics.EtherCatMasterX001.EtherCatMaster_HMI)
    Frame (13,284 262x172)
        shows V_Module(HMI := MAIN.Machine.Station_2.PackMLBaseModule_HMI)
    Frame (293,284 262x172)
        shows V_Module(HMI := MAIN.Machine.Station_3.PackMLBaseModule_HMI)
    Frame (13,522 262x172)
        shows V_Module(HMI := MAIN.Machine.Station_1.PackMLBaseModule_HMI)
    Frame (293,579 262x172)
        shows V_Module(HMI := MAIN.MachineStation_6.PackMLBaseModule_HMI)
END_VISUALIZATION
